# EPICS autosave request: BPMApp/Db/BPMSP_settings.req
$(P)$(R)BPMMode
